FUNCTION_BLOCK FieldsToEventFilter (* Transform individual fields to an Arrowhead Event Filter type *)
  (* Standard: 61499-2; Description: Copyright (c) 2019 fortiss GmbH This program and the accompanying materials are made available under the terms of the Eclipse Public License 2.0 which is available at https://www.eclipse.org/legal/epl-2.0/ SPDX-License-Identifier: EPL-2.0 *)
  (* Version 1.0, 2019-09-17, Cabral, fortiss GmbH *)
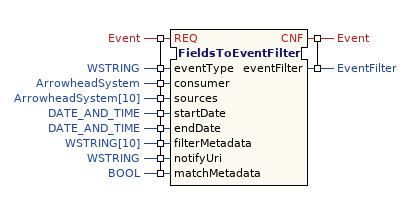
  EVENT_INPUT
    REQ WITH eventType, consumer, startDate, notifyUri, sources, endDate, filterMetadata, matchMetadata; (* Normal Execution Request *)
  END_EVENT
  EVENT_OUTPUT
    CNF WITH eventFilter; (* Execution Confirmation *)
  END_EVENT
  VAR_INPUT
    eventType : WSTRING; (* Event type, similar to topics in MQTT *)
    consumer : ArrowheadSystem; (* The Subscriber ArrowheadSystem, that will consume the new events *)
    sources : ARRAY [0..9] OF ArrowheadSystem; (* List of ArrowheadSystem the Subscriber wants to receive events from *)
    startDate : DATE_AND_TIME; (* If set, the Subscriber wants to receive events with timestamps after this date-time *)
    endDate : DATE_AND_TIME; (* If set, the Subscriber wants to receive events with timestamps before this date-time *)
    filterMetadata : ARRAY [0..9] OF WSTRING; (* Metadata about the events, which can be used for further filtering in format key=value *)
    notifyUri : WSTRING; (* The URL subpath where the Event Handler should sent the new events to *)
    matchMetadata : BOOL; (* Should the Event Handler filter events based on the metadata *)
  END_VAR
  VAR_OUTPUT
    eventFilter : EventFilter; (* Created Arrowhead event Filter *)
  END_VAR
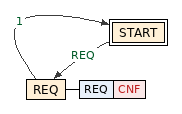
  EC_STATES
    START; (* Initial State *)
    REQ : REQ -> CNF;
  END_STATES
  EC_TRANSITIONS
    REQ TO START := 1;
    START TO REQ := REQ;
  END_TRANSITIONS
  ALGORITHM REQ IN ST:
VAR_TEMP
	i : INT;
END_VAR
;

i := 0;
eventFilter.eventType := eventType;
eventFilter.consumer := consumer;
eventFilter.startDate := startDate;
eventFilter.endDate := endDate;
eventFilter.notifyUri := notifyUri;
eventFilter.matchMetadata := matchMetadata;

WHILE i < 10 DO // looks like while is faster than FOR when exporting to cpp
	eventFilter.sources[i] := sources[i];
	eventFilter.filterMetadata[i] := filterMetadata[i];
	i := i + 1;
END_WHILE;
  END_ALGORITHM
END_FUNCTION_BLOCK
